{attribute 'c++_compatible'}
///Object base FB for all FB's
FUNCTION_BLOCK FB_Object IMPLEMENTS I_Object
VAR
    sName : STRING(50) := 'FB_Object'; //FB Name
    sVersion : STRING(8) := '1.0.0.0'; //FB Version
    bFirstPass : BOOL := FALSE; //First pass done
    bError : BOOL := FALSE; //Error
    nErrorID : DWORD := 0; //Error id
    aErrors : T_ErrorHistory; //Error history
END_VAR

///Add error to error history
METHOD PROTECTED AddError
VAR_INPUT
	nErrorID : DWORD; //Error ID
END_VAR
VAR
	nAddErrorLoop : INT;
END_VAR
FOR nAddErrorLoop := GVL_ObjectSetup.cErrorHistMax TO (GVL_ObjectSetup.cErrorHistMin + 1) BY -1 DO
	aErrors[nAddErrorLoop] := aErrors[nAddErrorLoop - 1];
END_FOR
aErrors[GVL_ObjectSetup.cErrorHistMin] := nErrorID;
END_METHOD

///Control, override to get cyclic task in FB
METHOD INTERNAL Control
VAR_INPUT
END_VAR
END_METHOD

//Cycle Task, do not override this methode cyclic code is placed in M_Control 
METHOD CycleTask
IF NOT(bFirstPass) THEN
    bFirstPass := Init() = GVL_HResultSuccess.cHR_SuccesDone;
    IF NOT(bFirstPass) THEN
        RETURN;
	END_IF
END_IF
Control();
END_METHOD

(*Error, do not implement property override*)
PROPERTY Error : BOOL
GET
Error := bError;
END_GET
END_PROPERTY

(*error id, do not implement property override*)
PROPERTY ErrorID : DWORD
GET
ErrorID := nErrorID;
END_GET
END_PROPERTY

(*Pointer to error history, do not implement property override*)
PROPERTY Errors : POINTER TO T_ErrorHistory
GET
Errors := ADR(aErrors);
END_GET
END_PROPERTY

METHOD FB_init : BOOL
VAR_INPUT
	bInitRetains : BOOL; // if TRUE, the retain variables are initialized (warm start / cold start)
	bInCopyCode : BOOL;  // if TRUE, the instance afterwards gets moved into the copy code (online change)
END_VAR
bFirstPass := FALSE;
END_METHOD

///Initialize FB, Override to do custom initialize, no need to call super
METHOD INTERNAL Init : HRESULT
Init := GVL_HResultSuccess.cHR_SuccesDone;
END_METHOD

(*Name, do not implement property override*)
PROPERTY Name : STRING(50)
GET
Name := sName;
END_GET
END_PROPERTY

(*Reset error, allways call super*)
METHOD Reset
bError := FALSE;
nErrorID := 0;
END_METHOD

///Set error on the Object and add entry to error history
METHOD PROTECTED SetError
VAR_INPUT
	nErrorID : DWORD; //Error ID
END_VAR
VAR
    nSetErrorLoop : INT;
END_VAR
IF NOT(bError) THEN
	bError := TRUE;
	THIS^.nErrorID := nErrorID;
	FOR nSetErrorLoop := GVL_ObjectSetup.cErrorHistMax TO (GVL_ObjectSetup.cErrorHistMin + 1) BY -1 DO
    	aErrors[nSetErrorLoop] := aErrors[nSetErrorLoop - 1];
	END_FOR
	aErrors[GVL_ObjectSetup.cErrorHistMin] := nErrorID;
END_IF
END_METHOD

(*Version,do not implement property override*)
PROPERTY Version : STRING(8)
GET
Version := sVersion;
END_GET
END_PROPERTY

END_FUNCTION_BLOCK

(* stored: Version 1.1.0.1, ProductVersion 3.1.4019.2
   POU FB_Object: Id {7ae2b3bc-6889-427a-82e4-66c1a0f4f97f}, SpecialFunc None
   Method AddError: Id {26aececa-6134-4ea0-b147-75cddd786a49}
   Method Control: Id {b1c46935-f116-4df7-8461-83771a2e39a0}
   Method CycleTask: Id {eb714de1-926f-48dc-8981-1ce3b30d9fbe}
   Property Error: Id {d41bc890-e3af-4a7c-8e60-f03a1c619e63}
   Get Get: Id {fafeed1c-814a-4256-ad02-fbf90e5e8080}
   Property ErrorID: Id {63ffb5b2-2ae5-4a47-86b8-36564ac6ed39}
   Get Get: Id {5fa2b1a1-1e53-40b1-ae8d-24fcf2722b11}
   Property Errors: Id {fcbaa8a8-a2ef-4477-8ff4-d26aef6ce2a5}
   Get Get: Id {1c8fbf77-dd85-40e9-bedf-41f1ba55588a}
   Method FB_init: Id {3ab89805-0d3a-421a-8ebd-105e5791755c}
   Method Init: Id {4237cb80-d346-4a7c-938a-6d6c8c793f75}
   Property Name: Id {e3a4abb1-c213-4331-ae82-93a6832e0b2b}
   Get Get: Id {19fd6a49-162e-45e7-8066-bac017555338}
   Method Reset: Id {9560225a-1cab-4c8f-9ae8-4c6933de2dbc}
   Method SetError: Id {f7b289ae-e020-441f-a57b-6988eb02710a}
   Property Version: Id {41ae7693-4c80-4a34-85a8-401771f8ba14}
   Get Get: Id {d66ac97e-e833-4f41-bc32-7299379a9627} *)
